# EPICS autosave request: linkamT96App/Db/LinkamVacuum_settings.req
$(P):STARTVAC.VAL
$(P):VACUUM:SET.VAL
$(P):VACUUM.SCAN
$(P):PRESSURE.SCAN
$(P):VACUUM:UNIT:SET.VAL
$(P):VACUUM:UNIT.SCAN
